{attribute 'qualified_only'}
{attribute 'strict'}
TYPE eERROR :
(
	NO_ERROR := 0, //Defined operation was executed successfully
	HOMING_METHOD_INACTIVE:=1,//NO homing method selected 
	AXIS_NOT_ENABLED:=2,//Axis is not enabled 
	WRONG_MODE:=3,//Wrong mode of operation input 
	NO_DEVICE_LINK:=4//ModeOfOperation output variable is not linked in device config  
);
END_TYPE

(* stored: Version 1.1.0.1, ProductVersion 3.1.4024.6
   EnumerationTextList eERROR: Id {abc2949a-f95b-45ab-987b-ef824813a646} *)
